FUNCTION_BLOCK AE_EVENT_TO_E (* Composite FB for convert EVENT to AE *)
  (* Standard: 61499-2; Description: Copyright (c) 2024 HR Agrartechnik GmbH This program and the accompanying materials are made available under the terms of the Eclipse Public License 2.0 which is available at https://www.eclipse.org/legal/epl-2.0/ SPDX-License-Identifier: EPL-2.0 *)
  (* Version 1.0, 2024-04-24, Franz Höpfinger, HR Agrartechnik GmbH *)
  PACKAGE adapter::conversion::unidirectional;
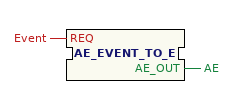
  EVENT_INPUT
    REQ; (* Request to Adapter *)
  END_EVENT
  PLUGS
    AE_OUT : adapter::types::unidirectional::AE; (* Adapter Output *)
  END_PLUGS
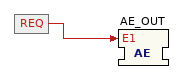
  EVENT_CONNECTIONS
    REQ TO AE_OUT.E1;
  END_CONNECTIONS
END_FUNCTION_BLOCK
